FUNCTION_BLOCK edgeneg
VAR_INPUT
	IN	: BOOL;
END_VAR
VAR_OUTPUT
	Q	: BOOL;
END_VAR
VAR
END_VAR

END_FUNCTION_BLOCK

(* stored: Version 1.1.0.1, ProductVersion 3.1.4024.12
   POU edgeneg: Id {9678accc-1061-4c06-b19f-5f237a6e99c0}, SpecialFunc None *)
